Fanuc KAREL source: kx00016.KL

-- PROVISIONAL review KL for V940-1; original PC SHA256 1513aa5fe9c01c36f84a2aa571e4a48aab090c86d3f0f4df5cd8c4401604d5eb
-- Incomplete behavior may be omitted. Consult companion uncertainty JSON. Do not deploy.
PROGRAM KX00016
%NOLOCKGROUP
VAR
  I : INTEGER
  J : INTEGER
  B : BOOLEAN
  F : FILE
  S : STRING[80]
-- UNRESOLVED_DECL P type=000102
BEGIN
  -- V9_ZERO_TABLE_METADATA_HINT layout=0001; no indexed target words; source/name/runtime held
  -- UNRESOLVED_PC offsets 5-7; opcodes 9D,0D
  -- UNRESOLVED_PC offsets 12-16; opcodes 7F
END KX00016
